{attribute 'qualified_only'}
VAR_GLOBAL CONSTANT
	axisNum:INT:=3;
END_VAR

(* stored: Version 1.1.0.1, ProductVersion 3.1.4024.0
   GVL GVL_APP: Id {0f050111-7af3-4866-869b-8f17050efbbe} *)
